FUNCTION_BLOCK X2Y2_J2_test (* Compute X^2-Y^2 in Java with explicit CNF invocation *)
  (* Standard: 61499-1 *)
  (* Version 0.0, 2009-05-12, JHC, Holobloc Inc, Modified from X2Y2_J as an example of CNF invocation. *)
  (* Compiler header: package fb.rt.student; *)
  (* Compiler Java Sun JDK 1.6.0 *)
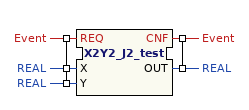
  EVENT_INPUT
    REQ WITH X, Y;
  END_EVENT
  EVENT_OUTPUT
    CNF WITH OUT;
  END_EVENT
  VAR_INPUT
    X : REAL;
    Y : REAL;
  END_VAR
  VAR_OUTPUT
    OUT : REAL;
  END_VAR
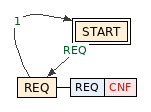
  EC_STATES
    START; (* Initial State *)
    REQ : REQ -> CNF; (* Normal execution *)
  END_STATES
  EC_TRANSITIONS
    START TO REQ := REQ;
    REQ TO START := 1;
  END_TRANSITIONS
  ALGORITHM REQ IN Java:
OUT.value = (X.value-Y.value)*(X.value+Y.value);
  END_ALGORITHM
END_FUNCTION_BLOCK
